FUNCTION_BLOCK E_SWITCH_CLOCK (* Switches between EI1 and EI2 to trigger EO (starting with EI1) *)
  (* Standard: 61499-2 *)
  (* Version 0.0, 2017-06-12, Marc Jakobi, HTW Berlin *)
  (* Version 1.0, 2016-05-26, AZ, fortiss GmbH *)
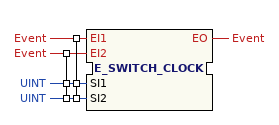
  EVENT_INPUT
    EI1 WITH SI1, SI2; (* Input event 1 *)
    EI2 WITH SI1, SI2; (* Input event 2 *)
  END_EVENT
  EVENT_OUTPUT
    EO; (* Output event *)
  END_EVENT
  VAR_INPUT
    SI1 : UINT; (* Switch to E2 after SI1 arrivals of EI1 *)
    SI2 : UINT; (* Switch to E1 after SI1 arrivals of EI2 *)
  END_VAR
  VAR
    CI1 : UINT; (* Counter for EI1 *)
    CI2 : UINT; (* Counter for EI2 *)
    EI2ACTIVE : BOOL; (* TRUE if EI2 is active *)
  END_VAR
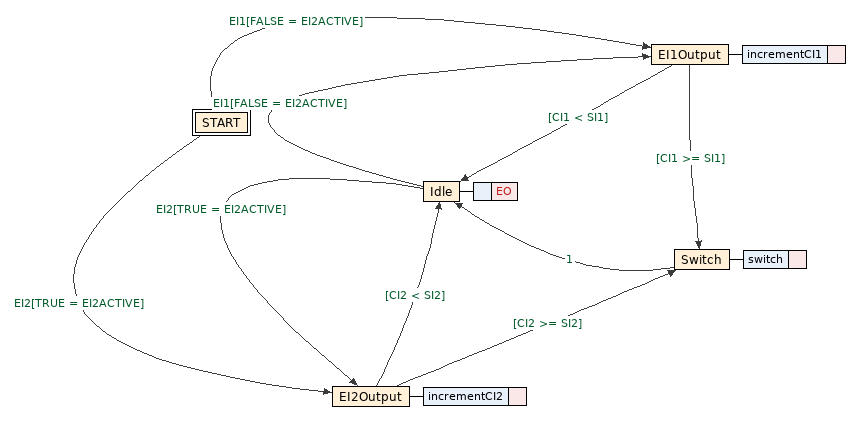
  EC_STATES
    START; (* Initial State *)
    EI1Output : incrementCI1; (* Normal execution *)
    EI2Output : incrementCI2;
    Switch : switch;
    Idle : -> EO;
  END_STATES
  EC_TRANSITIONS
    START TO EI1Output := EI1[FALSE = EI2ACTIVE];
    START TO EI2Output := EI2[TRUE = EI2ACTIVE];
    EI2Output TO Switch := [CI2 >= SI2];
    EI1Output TO Switch := [CI1 >= SI1];
    Switch TO Idle := 1;
    EI1Output TO Idle := [CI1 < SI1];
    EI2Output TO Idle := [CI2 < SI2];
    Idle TO EI1Output := EI1[FALSE = EI2ACTIVE];
    Idle TO EI2Output := EI2[TRUE = EI2ACTIVE];
  END_TRANSITIONS
  ALGORITHM incrementCI1 IN ST: (* Increments CI1 counter by 1 *)
CI1 := CI1 + 1;
  END_ALGORITHM
  ALGORITHM incrementCI2 IN ST: (* Increments CI2 counter by 1 *)
CI2 := CI2 + 1;
  END_ALGORITHM
  ALGORITHM switch IN ST: (* Resets counters to 0 and switches active event *)
CI1 := 0;
CI2 := 0;
EI2ACTIVE := NOT EI2ACTIVE;
  END_ALGORITHM
  (* Service left interface/right interface: Switches between EI1 and EI2 to trigger EO (starting with EI1) *)
END_FUNCTION_BLOCK
